# EPICS autosave request: GALILMUL/iocBoot/iocGALILMUL-IOC-01/GALIL_01_positions.req
file "GALIL_controller_positions.req" "P=$(P),CCP=$(CCP)"
